PROGRAM ClockPulse10ms
VAR
END_VAR

IF bClockPulse_10ms THEN
	bClockPulse_10ms := FALSE;
ELSE 
	bClockPulse_10ms := TRUE;	
END_IF

END_PROGRAM

(* stored: Version 1.1.0.1, ProductVersion 3.1.4024.12
   POU ClockPulse10ms: Id {0d96e69d-720a-4aca-abaa-8782f8daae15}, SpecialFunc None *)
